FUNCTION_BLOCK PicAlpha EXTENDS BaseCarrier
VAR_INPUT
END_VAR
VAR_OUTPUT
	o_VacuumGripper: VacuumGripper;
	o_MonostableCylinder: MonostableCylinder;
	o_Distance: INT := 50;
END_VAR
VAR
	m_PresenceSensorPosition1: PresenceSensor;
	m_PresenceSensorPosition2: PresenceSensor;
	m_PresenceSensorPosition3: PresenceSensor;
	m_PresenceSensorPosition4: PresenceSensor;

END_VAR

METHOD METH_CarrierBackward : BOOL
VAR_INPUT
END_VAR
Motor.ACT_TurnCounterclockwise();

IF m_PresenceSensorPosition1.Value THEN
	o_Distance := 0;
ELSIF m_PresenceSensorPosition2.Value THEN
	o_Distance := 10;
ELSIF m_PresenceSensorPosition3.Value THEN
	o_Distance := 50;
ELSIF m_PresenceSensorPosition4.Value THEN
	o_Distance := 100;
END_IF
END_METHOD

METHOD METH_CarrierForward : BOOL
VAR_INPUT
END_VAR
Motor.ACT_TurnClockwise();

IF m_PresenceSensorPosition1.Value THEN
	o_Distance := 0;
ELSIF m_PresenceSensorPosition2.Value THEN
	o_Distance := 10;
ELSIF m_PresenceSensorPosition3.Value THEN
	o_Distance := 50;
ELSIF m_PresenceSensorPosition4.Value THEN
	o_Distance := 100;
END_IF
END_METHOD

METHOD METH_CarrierStop : BOOL
VAR_INPUT
END_VAR
Motor.ACT_Stop();
END_METHOD

PROPERTY PresenceSensorPosition1Value : BOOL
GET
PresenceSensorPosition1Value := m_PresenceSensorPosition1.Value;
END_GET
END_PROPERTY

PROPERTY PresenceSensorPosition2Value : BOOL
GET
PresenceSensorPosition2Value := m_PresenceSensorPosition2.Value;
END_GET
END_PROPERTY

PROPERTY PresenceSensorPosition3Value : BOOL
GET
PresenceSensorPosition3Value := m_PresenceSensorPosition3.Value;
END_GET
END_PROPERTY

PROPERTY PresenceSensorPosition4Value : BOOL
GET
PresenceSensorPosition4Value := m_PresenceSensorPosition4.Value;
END_GET
END_PROPERTY

END_FUNCTION_BLOCK

(* stored: Version 1.1.0.1
   POU PicAlpha: Id {03071636-a184-4bb1-a2c6-5d782284ea47}, SpecialFunc None
   Method METH_CarrierBackward: Id {907c736b-471f-4c74-bb3c-e3f968d7c191}
   Method METH_CarrierForward: Id {b302867a-e7ad-427b-9cf6-40df8a3979e2}
   Method METH_CarrierStop: Id {50d58e4d-322a-4c5a-9c9f-f777502b5be9}
   Property PresenceSensorPosition1Value: Id {e96c7794-5ac9-4be1-abc7-0d40fe8317b5}
   Get Get: Id {d0cbf5aa-6d0a-4a0b-9728-cb6ec8b22d99}
   Property PresenceSensorPosition2Value: Id {f997094f-9bfe-449c-9329-ab9fba3c55f6}
   Get Get: Id {d8daaf04-dc2b-4c2c-b9ef-374b252cc252}
   Property PresenceSensorPosition3Value: Id {4431b3d5-9c0c-4905-9867-3fd8dfca0c86}
   Get Get: Id {ffe2ac42-5a84-47a8-bbd9-f5dbba64c46d}
   Property PresenceSensorPosition4Value: Id {19ce0e74-d2a8-41d6-8ed0-dafc504ad661}
   Get Get: Id {7d2b915d-f247-4c47-a486-8dc58545ecc9} *)
